TYPE ST_CFG_ProBoxElementMotor EXTENDS ST_CFG_ProBoxElementBase :
STRUCT
END_STRUCT
END_TYPE

(* stored: Version 1.1.0.1, ProductVersion 3.1.4024.9
   DUT ST_CFG_ProBoxElementMotor: Id {fea09d2f-aed0-42c4-bb47-01f342c8ed0b} *)
